TYPE PickPars_typ :
STRUCT
	
	Place		: Vector3Position_typ;
	Elevator	: Vector3Position_typ;
	ConvXTS 	: Vector3Position_typ;
	HomePos		: Vector3Position_typ;
	DumpPos		: Vector3Position_typ;
	LoadTime	: TIME;
	UnloadTime	: TIME;

END_STRUCT
END_TYPE

(* stored: Version 1.1.0.1, ProductVersion 3.1.4024.11
   DUT PickPars_typ: Id {d087dfb7-ff8c-4aaf-b542-399780117ac0} *)
